{attribute 'GeneratedUsingTerminal: EK1100-0000-0018'}
{attribute addProperty BoxType "EK1100-0000-0018"}
{attribute addProperty Id "Term_10_EK1122Term_10_EK1122_152EB6C21211Term_34_EL3403EL3403_812980A665Term_35_EL6001EL6001_0DE01E7E61Term_36_EL3024EL3024_C6E76B5A40Term_33_EL9011EL9011_D65D3D320"}
{attribute addProperty CRC "230948961"}
{attribute addProperty Size "1377"}
{attribute addProperty Name "Term 9 (EK1100)"}
TYPE Term_9_EK1100_0DC40061 EXTENDS EK1100_1FC0878B :
STRUCT
	{attribute addProperty Name "Term 10 (EK1122)"}
	{attribute addProperty PreviousPort "Term 9 (EK1100) : B"}
	{attribute addProperty SyncUnit "default"}
	Term_10_EK1122 : Term_10_EK1122_152EB6C2;
	{attribute addProperty Name "Term 34 (EL3403)"}
	{attribute addProperty PreviousPort "Term 10 (EK1122) : C"}
	{attribute addProperty SyncUnit "Row_0"}
	Term_34_EL3403 : EL3403_812980A6;
	{attribute addProperty Name "Term 35 (EL6001)"}
	{attribute addProperty PreviousPort "Term 34 (EL3403) : B"}
	{attribute addProperty SyncUnit "Row_0"}
	Term_35_EL6001 : EL6001_0DE01E7E;
	{attribute addProperty Name "Term 36 (EL3024)"}
	{attribute addProperty PreviousPort "Term 35 (EL6001) : B"}
	{attribute addProperty SyncUnit "Row_0"}
	Term_36_EL3024 : EL3024_C6E76B5A;
	{attribute addProperty Name "Term 33 (EL9011)"}
	{attribute addProperty PreviousPort "Term 36 (EL3024) : B"}
	{attribute addProperty SyncUnit "default"}
	Term_33_EL9011 : EL9011_D65D3D32;
END_STRUCT
END_TYPE

(* stored: Version 1.2.0.0, ProductVersion 3.1.4024.11
   DUT Term_9_EK1100_0DC40061: Id {f480b48e-6d8f-4c95-92ca-ae061cafeb44} *)
